# EPICS autosave request: iocBoot/generic_motors_ioc/dbSave/MO_Ps_.req
%
% BURT Request File
%
% $(P)MO:Ps:  Monochromator Positioning (alignment)
%

file assy.req ASSY=$(P)MO:Ps
file mtr1.req MTR1=$(P)MO:mz
file mtr1.req MTR1=$(P)MO:my
file drv1.req DRV1=$(P)MO:Z
file drv1.req DRV1=$(P)MO:Y
